KUKA KRL program: Bolge_2_Palet_Ort.src, Bolge_2_Palet_Ort.dat

--- Bolge_2_Palet_Ort.src ---
&ACCESS RVP
&REL 71
&PARAM DISKPATH = KRC:\R1\Program\Sub_Rutinler
DEF  Bolge_2_Palet_Ort ( )
;FOLD INI;%{PE}
  ;FOLD BASISTECH INI
    GLOBAL INTERRUPT DECL 3 WHEN $STOPMESS==TRUE DO IR_STOPM ( )
    INTERRUPT ON 3
    BAS (#INITMOV,0 )
  ;ENDFOLD (BASISTECH INI)
  ;FOLD USER INI
    ;Make your modifications here

  ;ENDFOLD (USER INI)
;ENDFOLD (INI)



;;FOLD PTP B2_MASTER CONT Vel=100 % PDAT2 Tool[1]:Gripper Base[0] ;%{PE}
;;FOLD Parameters ;%{h}
;;Params IlfProvider=kukaroboter.basistech.inlineforms.movement.old; Kuka.IsGlobalPoint=False; Kuka.PointName=B2_MASTER; Kuka.BlendingEnabled=True; Kuka.MoveDataPtpName=PDAT2; Kuka.VelocityPtp=100; Kuka.CurrentCDSetIndex=0; Kuka.MovementParameterFieldEnabled=True; IlfCommand=PTP
;;ENDFOLD
;$BWDSTART = FALSE
;PDAT_ACT = PPDAT2
;FDAT_ACT = FB2_MASTER
;BAS(#PTP_PARAMS, 100.0)
;SET_CD_PARAMS (0)
;PTP XB2_MASTER C_Dis
;;ENDFOLD


PaletMasterX=1020
PaletMasterY=1020

Base_Data[2]=Frame_Donustur(XB2_MASTER)
BASE_DATA[2].x=BASE_DATA[2].x+(PaletMasterX/2)
BASE_DATA[2].Y=BASE_DATA[2].Y-(PaletMasterY/2)

      IF (ParcaUzunluk<=1500)THEN

         BASE_DATA[2].x=BASE_DATA[2].x-(PaletUzunluk/2)
         BASE_DATA[2].Y=BASE_DATA[2].Y+(PaletGenislik/2)

      ENDIF

      IF (ParcaUzunluk>=1600) AND (ParcaUzunluk<=3000) THEN

         BASE_DATA[2].x=BASE_DATA[2].x-(PaletUzunluk/2)
         BASE_DATA[2].Y=BASE_DATA[2].Y+(PaletGenislik/2)

      ENDIF

END
DEFFCT FRAME Frame_Donustur(e6GeciciPos:IN)
   ;FOLD  Tanimlamalar
      DECL E6POS e6GeciciPos
      DECL FRAME ReturnFrame
   ;ENDFOLD
   ReturnFrame=$Nullframe
   ReturnFrame.X=e6GeciciPos.X
   ReturnFrame.Y=e6GeciciPos.Y
   ReturnFrame.Z=e6GeciciPos.Z
   ReturnFrame.A=e6GeciciPos.A
   ReturnFrame.B=e6GeciciPos.B
   ReturnFrame.C=e6GeciciPos.C
   RETURN ReturnFrame
ENDFCT

--- Bolge_2_Palet_Ort.dat ---
&ACCESS RVP1
&REL 71
&PARAM DISKPATH = KRC:\R1\Program\Sub_Rutinler
DEFDAT  BOLGE_2_PALET_ORT
;FOLD EXTERNAL DECLARATIONS;%{PE}%MKUKATPBASIS,%CEXT,%VCOMMON,%P
;FOLD BASISTECH EXT;%{PE}%MKUKATPBASIS,%CEXT,%VEXT,%P
EXT  BAS (BAS_COMMAND  :IN,REAL  :IN )
DECL INT SUCCESS
;ENDFOLD (BASISTECH EXT)
;FOLD USER EXT;%{E}%MKUKATPUSER,%CEXT,%VEXT,%P
;Make your modifications here

;ENDFOLD (USER EXT)
;ENDFOLD (EXTERNAL DECLARATIONS)
DECL PDAT PPDAT1={VEL 100.000,ACC 100.000,APO_DIST 500.000,APO_MODE #CDIS,GEAR_JERK 100.000,EXAX_IGN 0}
DECL FDAT FB1_Master_1={TOOL_NO 1,BASE_NO 0,IPO_FRAME #BASE,POINT2[] " "}
DECL E6POS XB2_MASTER={X -783.939758,Y 1836.30701,Z -1215.86841,A -0.181200683,B -2.63909937E-14,C -3.09510859E-12,S 6,T 51,E1 0.0,E2 0.0,E3 0.0,E4 0.0,E5 0.0,E6 0.0}
DECL FDAT FB2_MASTER={TOOL_NO 1,BASE_NO 0,IPO_FRAME #BASE,POINT2[] " "}
DECL PDAT PPDAT2={VEL 100.000,ACC 100.000,APO_DIST 500.000,APO_MODE #CDIS,GEAR_JERK 100.000,EXAX_IGN 0}
DECL MODULEPARAM_T LAST_TP_PARAMS={PARAMS[] "Kuka.PointName=B3_MASTERtet; Kuka.FrameData.base_no=0; Kuka.FrameData.tool_no=1; Kuka.FrameData.ipo_frame=#BASE; Kuka.FrameData.point2=; Kuka.isglobalpoint=False; Kuka.MoveDataPtpName=PDAT2; Kuka.MovementDataPdat.apo_mode=#CDIS; Kuka.MovementDataPdat.apo_dist=500; Kuka.MovementData.vel=0.1; Kuka.MovementData.acc=100; Kuka.MovementData.exax_ign=0; Kuka.VelocityPtp=100; Kuka.BlendingEnabled=True; Kuka.APXEnabled=False; Kuka.CurrentCDSetIndex=0; Kuka.MoveDataName=CPDAT1; Kuka.MovementData.cb={AUX_PT {ORI #CONSIDER,E1 #CONSIDER,E2 #CONSIDER,E3 #CONSIDER,E4 #CONSIDER,E5 #CONSIDER,E6 #CONSIDER},TARGET_PT {ORI #INTERPOLATE,E1 #INTERPOLATE,E2 #INTERPOLATE,E3 #INTERPOLATE,E4 #INTERPOLATE,E5 #INTERPOLATE,E6 #INTERPOLATE}}; Kuka.MovementData.apo_fac=50; Kuka.MovementData.apo_dist=500; Kuka.MovementData.axis_acc=100; Kuka.MovementData.axis_vel=100; Kuka.MovementData.circ_typ=#BASE; Kuka.MovementData.jerk_fac=50; Kuka.MovementData.ori_typ=#VAR; Kuka.VelocityPath=0.1"}
DECL E6POS XB3_MASTERtet={X -955.559,Y 1787.95337,Z -1211.09766,A -0.418937892,B 3.83629760E-13,C -2.32866417E-12,S 6,T 59,E1 0.0,E2 0.0,E3 0.0,E4 0.0,E5 0.0,E6 0.0}
DECL FDAT FB3_MASTERtet={TOOL_NO 1,BASE_NO 0,IPO_FRAME #BASE,POINT2[] " "}
DECL LDAT LCPDAT1={VEL 0.100000,ACC 100.000,APO_DIST 500.000,APO_FAC 50.0000,AXIS_VEL 100.000,AXIS_ACC 100.000,ORI_TYP #VAR,CIRC_TYP #BASE,JERK_FAC 50.0000,GEAR_JERK 100.000,EXAX_IGN 0,CB {AUX_PT {ORI #CONSIDER,E1 #CONSIDER,E2 #CONSIDER,E3 #CONSIDER,E4 #CONSIDER,E5 #CONSIDER,E6 #CONSIDER},TARGET_PT {ORI #INTERPOLATE,E1 #INTERPOLATE,E2 #INTERPOLATE,E3 #INTERPOLATE,E4 #INTERPOLATE,E5 #INTERPOLATE,E6 #INTERPOLATE}}}
ENDDAT
